// Mitsubishi GX Works2 project: 240926_공급가공2   PLC: Q03UDV

PROGRAM MAIN
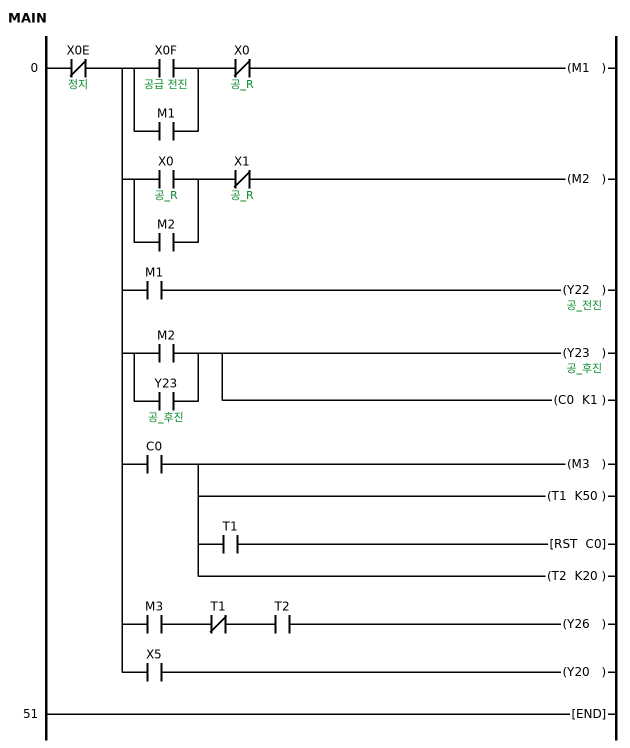
0     LDI     X0E  ; 정지
      MPS
      LD      X0F  ; 공급 전진
      OR      M1
      ANB
      ANI     X0  ; 공_R
      OUT     M1
      MRD
      LD      X0  ; 공_R
      OR      M2
      ANB
      ANI     X1  ; 공_R
      OUT     M2
      MRD
      AND     M1
      OUT     Y22  ; 공_전진
      MRD
      LD      M2
      OR      Y23  ; 공_후진
      ANB
      OUT     Y23  ; 공_후진
      OUT     C0 K1
      MRD
      AND     C0
      OUT     M3
      OUT     T1 K50
      MPS
      AND     T1
      RST     C0
      MPP
      OUT     T2 K20
      MRD
      AND     M3
      ANI     T1
      AND     T2
      OUT     Y26
      MPP
      AND     X5
      OUT     Y20
51    END
END_PROGRAM

// device comments not shown above
X4  ; 가공_F
Y24  ; 공_후진
